FUNCTION_BLOCK FB_InterfaceProfibus IMPLEMENTS ITF_Cell
VAR_INPUT

END_VAR
VAR_OUTPUT
END_VAR

VAR
	// Ausgang :engine          AT %IX0.0:        BOOL; 
//Eingänge
//A5Q_Bestuckung AT %QX27.4 : BOOL;
//A5Q_Startfreigabe AT %QX27.5 : BOOL;
//A5Q_Entnahme AT %QX27.6 : BOOL;
//A5Q_Standby AT %QX27.7 : BOOL;
//A5Q_NOT_Aus_Befehl AT %QX28.0 : BOOL;

//INPUTS  A5 Station Variabel : 5V Von Arduino

//A5I_Bestuckbereit_o1 AT %IX43.2 : BOOL;  
//A5I_Arbeitet_o2 AT %IX43.3 : BOOL;
//A5I_Fertig_o3 AT %IX43.4 : BOOL;
//A5I_Storung_o5 AT %IX43.5 : BOOL;
//A5I_NOT_Halt_o6 AT %IX43.6 : BOOL;
//A5I_Pro_Standby_o7 AT %IX43.7 : BOOL;
//A5I_Pro_Standby_o8 AT %IX44.0 : BOOL;
/////////////////////////////////////////////////////////////////////////////////////////////////////////////////
//*Hami* boolesche Eingänge und Ausgänge als innere Variable deklarieren 

//*Hami* innere Eingänge
m_bEmergencyOff  : BOOL; 
m_bEmergencyStop : BOOL;
m_bFinished : BOOL;
m_bRunning : BOOL;
m_bLoadPos  : BOOL; 
m_bUnloadPos  : BOOL; 
m_bStandby : BOOL;
m_bStartable : BOOL;
m_bSoftError  : BOOL;

//*Hami* innere Ausgänge
m_bToEmergencyOff  : BOOL;
m_bToEmergencyStop  : BOOL;
m_bMoveToLoadPos  : BOOL;
m_bMoveToUnloadPos : BOOL;
m_bToStandby  : BOOL;
m_bStart  : BOOL;

//*HAMI* Eingäng und Ausgäng in Form UINT deklarieren zum anpassen Profibus_Dateien
//*HAMI* Die beide müssen zu ProfibusKlemme gelinkt werden

m_wProfibusDataWord AT %I*  : UINT; 
m_wToProfibusDataWord AT %Q*  : UINT;

//*HAMI* Hilf_FBs Deklarieren (Konvertor)

fbBoolToWord : FB_Bool_To_Word;
fbWordToBool : FB_Word_To_Bool;
//*HAMI* Variable für Konvertor FBs ( FB_Bool_to_Word und FB_Word_to_bool )
//*HAMI* i_arrayOfBool Eingänge q_arrayOfBool Ausgänge
i_arrayOfBool : ARRAY [0..15] OF BOOL;
q_arrayOfBool : ARRAY [0..15] OF BOOL;
//*Hami physikalische Eingänge und Ausgänge von Profibus werden drin geschrieben *
i_DataWord : UINT ;
q_DataWord : UINT ;
/////////////////////////////////////////////////////////////////////////////////////////////////////////////////


END_VAR

/////////////////////////////////////////////////////////////////////////////////////////////////////////////////
//*Hami* Aufruf von Hilf_FBs (Konvertor) 
fbBoolToWord();
fbWordToBool();


//hier Wird Mit Hilfe Von Funktion Blocks ( FB_Bool_to_Word und FB_Word_to_bool ) eingänge und Ausgänge angepasst

// Eingänge von Zelle To Bool
i_DataWord := m_wProfibusDataWord ;  //*Hami* Eingang von Profibus in einem hilfsvariabel schreiben
fbWordToBool.i_Word := i_DataWord ; //*Hami* Eingang von Profibus in Eingang von FB_WordToBool schreiben 
i_arrayOfBool :=fbWordToBool.o_Bool ; //*Hami* Ausgang von FB_WordToBool in ein Array of Bool Schreiben 


//*Hami* jeder Index von Array wurde gleich innere Eingänge gestellt 
m_bEmergencyOff := i_arrayOfBool[0];
m_bEmergencyStop := i_arrayOfBool[1]; 
m_bFinished := i_arrayOfBool[2];
m_bRunning := i_arrayOfBool[3];
m_bLoadPos := i_arrayOfBool[4]; 
m_bUnloadPos := i_arrayOfBool[5];   
m_bStandby := i_arrayOfBool[6];
m_bStartable := i_arrayOfBool[7];
m_bSoftError := i_arrayOfBool[8];

//*Hami* Ausgänge von Zelle To Array of Bool 

q_arrayOfBool[0]:= m_bToEmergencyOff ;
q_arrayOfBool[1] := m_bToEmergencyStop;  
q_arrayOfBool[2] := m_bMoveToLoadPos;  
q_arrayOfBool[3] := m_bMoveToUnloadPos; 
q_arrayOfBool[4] := m_bToStandby;  
q_arrayOfBool[5] := m_bStart;

fbBoolToWord.i_Bool := q_arrayOfBool ;//*Hami* Array of Bool in Eingang von fbBoolToWord schreiben
q_DataWord := fbBoolToWord.o_Word ;  //*Hami*  Ausgang von FB_BoolToWord in einem Hilfsvariabel schreiben 
m_wToProfibusDataWord := q_DataWord ; //*Hami* Hilfsvariabel in Ausgang von Profibus Schreiben

/////////////////////////////////////////////////////////////////////////////////////////////////////////////////


// Logik des Interfaces in diesem Fall zurücksetzen der Ausgänge nach erreichen des Ziels 
// Aus Zustandsmaschine Löschen ggf. ??
//IF m_bEmergencyOff THEN
//m_bToEmergencyOff := FALSE;
//END_IF

//IF m_bEmergencyStop THEN
//m_bToEmergencyStop := FALSE;
//END_IF

IF m_bLoadPos THEN
	m_bMoveToLoadPos := FALSE;
END_IF

IF m_bUnloadPos THEN
	m_bMoveToUnloadPos := FALSE;
END_IF

IF m_bStandby THEN
	m_bToStandby := FALSE;
END_IF

IF m_bRunning THEN
	m_bStart := FALSE;
END_IF

METHOD GetEmergencyOff : BOOL
VAR_INPUT
END_VAR
GetEmergencyOff := m_bEmergencyOff;
END_METHOD

METHOD GetEmergencyStop : BOOL
VAR_INPUT
END_VAR
GetEmergencyStop := m_bEmergencyStop;
END_METHOD

METHOD GetFinished : BOOL
VAR_INPUT
END_VAR
GetFinished := m_bFinished;
END_METHOD

METHOD GetIsRunning : BOOL
VAR_INPUT
END_VAR
GetIsRunning := m_bRunning;
END_METHOD

METHOD GetLoadPos : BOOL
VAR_INPUT
END_VAR
GetLoadPos := m_bLoadPos;
END_METHOD

METHOD GetStandby : BOOL
VAR_INPUT
END_VAR
GetStandby := m_bStandby;
END_METHOD

METHOD GetStartable : BOOL
VAR_INPUT
END_VAR
GetStartable := m_bStartable;
END_METHOD

METHOD GetUnloadPos : BOOL
VAR_INPUT
END_VAR
GetUnloadPos := m_bUnloadPos;
END_METHOD

METHOD SetEmergencyOff : BOOL
VAR_INPUT
	b :BOOL;
END_VAR

m_bToEmergencyOff := b;
SetEmergencyOff:=b;
END_METHOD

METHOD SetEmergencyStop : BOOL
VAR_INPUT
	b :BOOL;
END_VAR
m_bToEmergencyStop :=b;

SetEmergencyStop := b;
END_METHOD

METHOD SetMoveToLoad : BOOL
VAR_INPUT
	b :BOOL;
END_VAR
m_bMoveToLoadPos := b;

SetMoveToLoad := b;
END_METHOD

METHOD SetMoveToUnload : BOOL
VAR_INPUT
	b :BOOL;
END_VAR
m_bMoveToUnloadPos := b;

SetMoveToUnload := b;
END_METHOD

METHOD SetStandby : BOOL
VAR_INPUT
	b :BOOL;
END_VAR
m_bToStandby := b;

SetStandby := b;
END_METHOD

METHOD SetStart : BOOL
VAR_INPUT
	b :BOOL;
END_VAR
m_bStart := b;

SetStart := b;
END_METHOD

END_FUNCTION_BLOCK

(* stored: Version 1.1.0.1, ProductVersion 3.1.4024.0
   POU FB_InterfaceProfibus: Id {40f5a530-d22d-4cda-b588-d4b13544feb3}, SpecialFunc None
   Method GetEmergencyOff: Id {9ddbebc1-2c22-496a-8486-87b6e9601fa8}
   Method GetEmergencyStop: Id {a1d6ad32-92e6-47f2-b12d-a15a4cd0551a}
   Method GetFinished: Id {9cfd8bcb-3945-4765-82c5-421db15b878e}
   Method GetIsRunning: Id {30836f67-2870-4726-a26f-d9b37208fbd2}
   Method GetLoadPos: Id {b1d79e76-efbb-41f3-a918-d6bad0c9ee1c}
   Method GetStandby: Id {f1a41f0e-c07a-4585-8fdd-392464027ec9}
   Method GetStartable: Id {c36847f7-5d90-4a0c-bb3a-c8f3e71f3aed}
   Method GetUnloadPos: Id {41bdac74-6578-4410-a0a5-201a9064dcf2}
   Method SetEmergencyOff: Id {fe6d2834-19fc-43a6-806f-fdc5e151cc99}
   Method SetEmergencyStop: Id {47c0fddc-0661-49f0-9e6e-88d23cb9bf6c}
   Method SetMoveToLoad: Id {88714bc4-724b-49ad-bca2-1a6e99f2b2bd}
   Method SetMoveToUnload: Id {f2e3f2df-41d9-421c-bb52-c8cc8dc2f937}
   Method SetStandby: Id {b783b6a9-e15f-4ec0-8540-101be5cc4bef}
   Method SetStart: Id {ac91bfb6-2035-4d8d-a468-f67ec83fb09a} *)
